FUNCTION_BLOCK FbCalculator
VAR_INPUT
END_VAR
VAR_OUTPUT
END_VAR
VAR
END_VAR

{attribute 'TcRpcEnable'}
METHOD PUBLIC Sum : LREAL
VAR_INPUT
    Input1 : LREAL;
    Input2 : LREAL;
END_VAR
Sum := Input1 + Input2;
END_METHOD

END_FUNCTION_BLOCK

(* stored: Version 1.1.0.1, ProductVersion 3.1.4024.9
   POU FbCalculator: Id {5c4ee6bf-053a-4b6e-bea8-c2082c4df868}, SpecialFunc None
   Method Sum: Id {84f43510-45e4-442c-bebe-0c11ddd676e0} *)
